(* Logix 5000 project; controller cal1615 1756-L62 rev 16.20; software revision 16.05; part 58 of 78 *)
(* tags used below, declared in another part *)
   FAULT : BOOL;   // Fault AFI
   HMI : BOOL;   // AFI HMI
   p01r09_pb_global_reset : BOOL;   // System Modes PB: Global Fault Reset
   p02_real_from_hmi : hmi_real;   // MOP HMI Iface Real from HMI
   p25_ai_amps : DINT;   // Tension Stand 2 Analog Input TS 2 Motor Current
   p25_ai_hz : DINT;   // Tension Stand 2 Analog Input TS 2 Motor Hertz
   p25_ai_rpm : REAL;
   p25_ai_speed : REAL;   // Tension Stand 2 Inputs Sufrace Speed [fpm]
   p25_ai_ts2_lc : REAL;   // System Metering Roll VFD Minimum Start Tension
   p25_ao_selected_speed : REAL;   // Tension Stand 2 VFD Selected Speed
   p25_ao_torque : REAL;
   p25_ao_vfd : REAL;
   p25_control_word : INT;
   p25_di_brake : BOOL;   // Tension Stand 2 Digital Input TS2 & Slitter Brake Temperature OK
   p25_di_therm : BOOL;   // Tension Stand 2 Digital Input Motor Temperature OK
   p25_di_ts2 : acs800_di_normal;   // Tension Stand 2 Digital Inputs VFD Inputs
   p25_dint_to_hmi : DINT[16];   // Tension Stand 2 Dint to HMI
   p25_real_to_hmi : REAL[112];   // Tension Stand 2 Real to HMI
   p25_status_word : INT;
   p25_ts2_gear_ratio : REAL;
   p25_ts2_roll_diameter_ft : REAL;
   p25_vfd_input_max : REAL;
   p25_vfd_input_min : REAL;
   p25_vfd_output_max : REAL;
   p25_vfd_output_min : REAL;
   p25r01 : routine;
   p25r03_vfd_out_scaling : SYS_SCP;
   p25r04 : routine;
   p25r04_speed_to_vfd_ts2_scp : SYS_SPEED_TO_VFD;   // Tension Stand 2 Outputs Speed to Tension Stand 2 VFD
   p25r04_timer_fault : TIMER[4];   // Tension Stand 2 Outputs Fault Dwell Timer
   p25r04_timer_warning : TIMER[4];   // Tension Stand 2 Outputs Warning Dwell Timer
   p25r05 : routine;
   p25r05_timer_fault : TIMER[4];   // Tension Stand 2 Dint to HMI Fault Dwell Timer
   p25r05_timer_warning : TIMER[4];   // Tension Stand 2 Dint to HMI Warning Dwell Time
   p25r06 : routine;
   p25r06_ave_lc : REAL;
   p25r06_lc_ave_ctrl : CONTROL;
   p25r06_lc_buffer : REAL[20];
   p25r06_lc_ctrl : CONTROL;
   p25r06_sample_timer : TIMER;
   p25r06_timer_fault : TIMER[4];   // Tension Stand 2 Real to HMI Fault Dwell Timer
   p25r06_timer_warning : TIMER[4];   // Tension Stand 2 Real to HMI Warning Dwell Timer
   p25r06_unload : REAL;
   p25r09_mode_jog : BOOL;   // Tension Stand 2 Modes Jog Mode
   p25r09_mode_run : BOOL;   // Tension Stand 2 Modes Run Mode
   p25r09_mode_thread : BOOL;   // Tension Stand 2 Modes Thread Mode
(* P25_Tension_Stand_2, continued *)

ROUTINE R04_Output   (* ladder *)
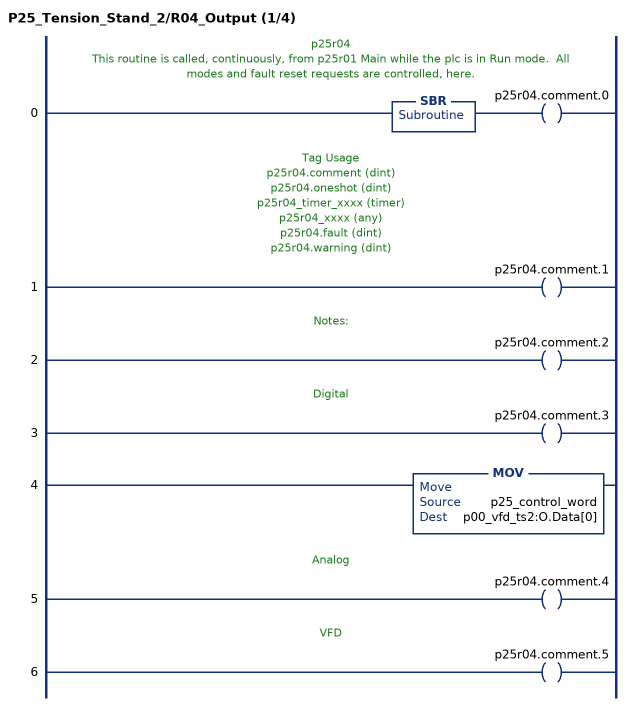
   // p25r04
   // This routine is called, continuously, from p25r01 Main while the plc is in Run mode.  All modes and fault reset requests are controlled, here.
   0: SBR()OTE(p25r04.comment.0);
   // Tag Usage
   // p25r04.comment (dint)
   // p25r04.oneshot (dint)
   // p25r04_timer_xxxx (timer)
   // p25r04_xxxx (any)
   // p25r04.fault (dint)
   // p25r04.warning (dint)
   1: OTE(p25r04.comment.1);
   // Notes:
   2: OTE(p25r04.comment.2);
   // Digital
   3: OTE(p25r04.comment.3);
   4: MOV(p25_control_word,p00_vfd_ts2:O.Data[0]);
   // Analog
   5: OTE(p25r04.comment.4);
   // VFD
   6: OTE(p25r04.comment.5);
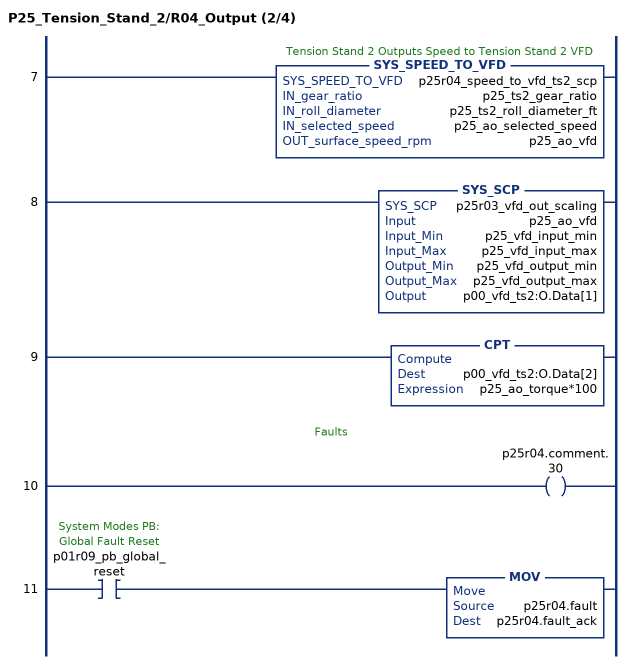
   7: SYS_SPEED_TO_VFD(p25r04_speed_to_vfd_ts2_scp,p25_ts2_gear_ratio,p25_ts2_roll_diameter_ft,p25_ao_selected_speed,p25_ao_vfd);
   8: SYS_SCP(p25r03_vfd_out_scaling,p25_ao_vfd,p25_vfd_input_min,p25_vfd_input_max,p25_vfd_output_min,p25_vfd_output_max,p00_vfd_ts2:O.Data[1]);
   9: CPT(p00_vfd_ts2:O.Data[2],p25_ao_torque*100);
   // Faults
   10: OTE(p25r04.comment.30);
   11: XIC(p01r09_pb_global_reset)MOV(p25r04.fault,p25r04.fault_ack);
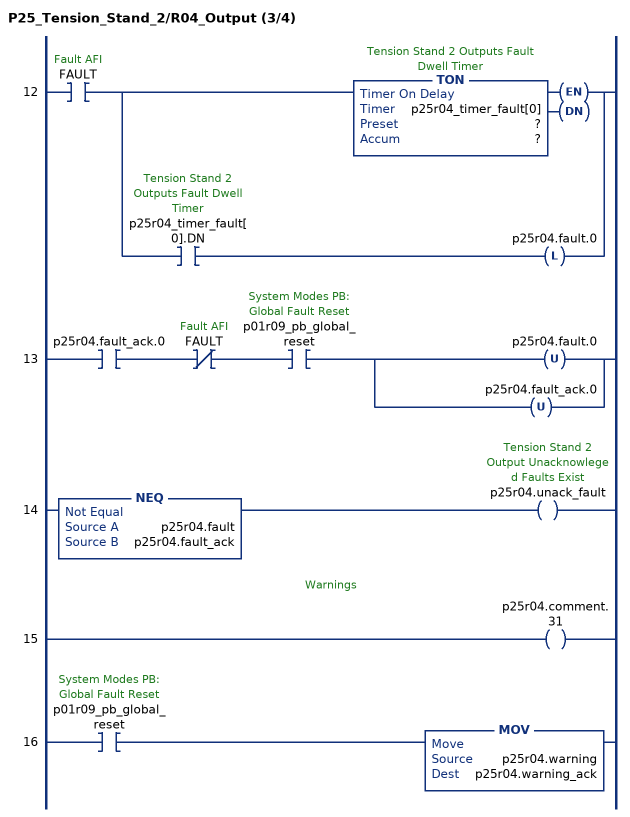
   12: XIC(FAULT)[TON(p25r04_timer_fault[0],?,?) ,XIC(p25r04_timer_fault[0].DN) OTL(p25r04.fault.0) ];
   13: XIC(p25r04.fault_ack.0)XIO(FAULT)XIC(p01r09_pb_global_reset)[OTU(p25r04.fault.0) ,OTU(p25r04.fault_ack.0) ];
   14: NEQ(p25r04.fault,p25r04.fault_ack)OTE(p25r04.unack_fault);
   // Warnings
   15: OTE(p25r04.comment.31);
   16: XIC(p01r09_pb_global_reset)MOV(p25r04.warning,p25r04.warning_ack);
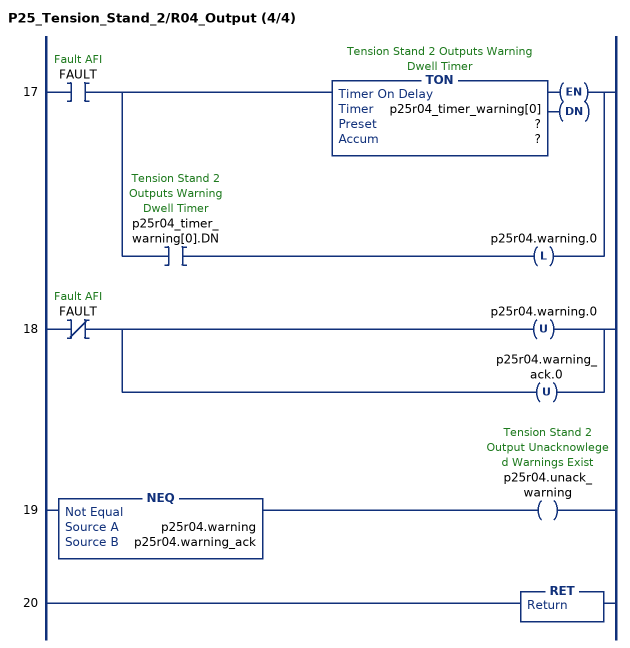
   17: XIC(FAULT)[TON(p25r04_timer_warning[0],?,?) ,XIC(p25r04_timer_warning[0].DN) OTL(p25r04.warning.0) ];
   18: XIO(FAULT)[OTU(p25r04.warning.0) ,OTU(p25r04.warning_ack.0) ];
   19: NEQ(p25r04.warning,p25r04.warning_ack)OTE(p25r04.unack_warning);
   20: RET();
END_ROUTINE

ROUTINE R05_Dint_to_HMI   (* ladder *)
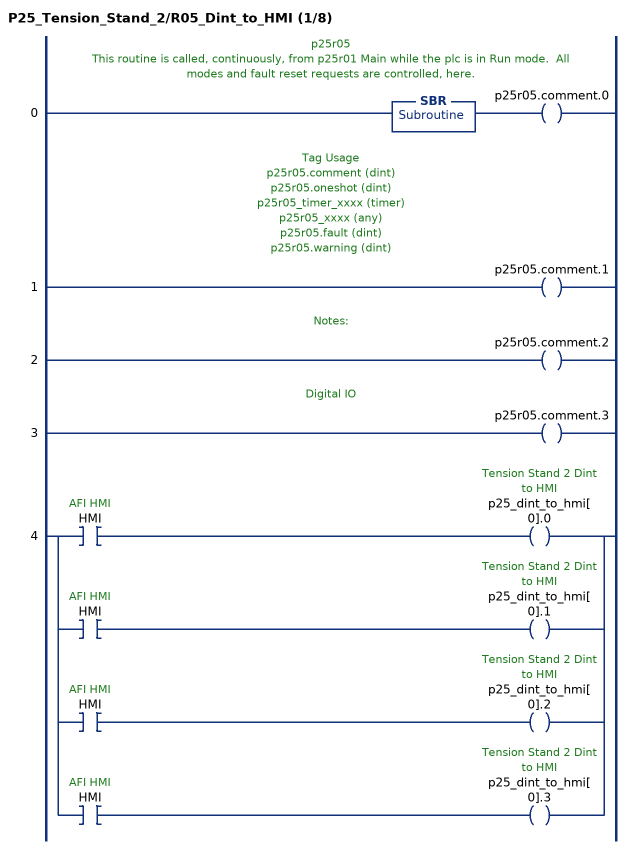
   // p25r05
   // This routine is called, continuously, from p25r01 Main while the plc is in Run mode.  All modes and fault reset requests are controlled, here.
   0: SBR()OTE(p25r05.comment.0);
   // Tag Usage
   // p25r05.comment (dint)
   // p25r05.oneshot (dint)
   // p25r05_timer_xxxx (timer)
   // p25r05_xxxx (any)
   // p25r05.fault (dint)
   // p25r05.warning (dint)
   1: OTE(p25r05.comment.1);
   // Notes:
   2: OTE(p25r05.comment.2);
   // Digital IO
   3: OTE(p25r05.comment.3);
   4: [XIC(HMI) OTE(p25_dint_to_hmi[0].0) ,XIC(HMI) OTE(p25_dint_to_hmi[0].1) ,XIC(HMI) OTE(p25_dint_to_hmi[0].2) ,XIC(HMI) OTE(p25_dint_to_hmi[0].3) ];
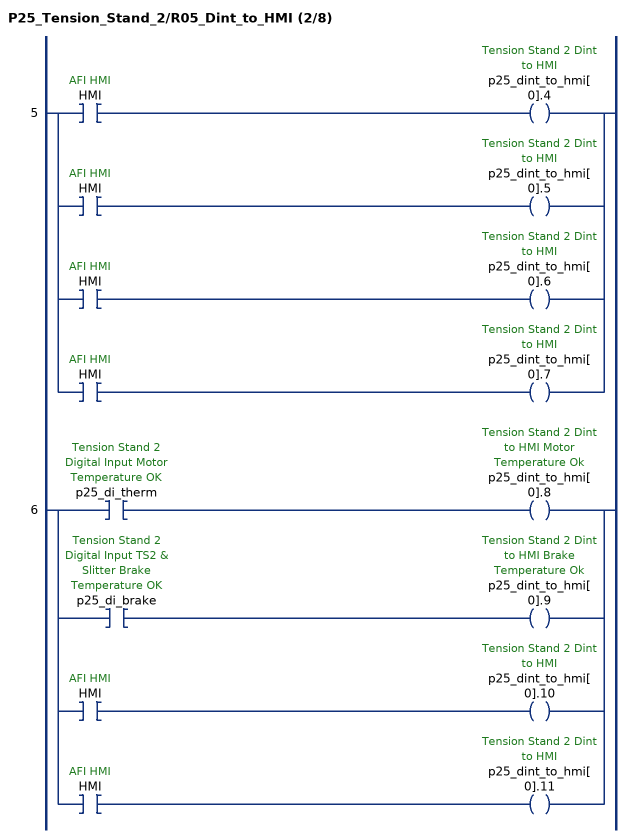
   5: [XIC(HMI) OTE(p25_dint_to_hmi[0].4) ,XIC(HMI) OTE(p25_dint_to_hmi[0].5) ,XIC(HMI) OTE(p25_dint_to_hmi[0].6) ,XIC(HMI) OTE(p25_dint_to_hmi[0].7) ];
   6: [XIC(p25_di_therm) OTE(p25_dint_to_hmi[0].8) ,XIC(p25_di_brake) OTE(p25_dint_to_hmi[0].9) ,XIC(HMI) OTE(p25_dint_to_hmi[0].10) ,XIC(HMI) OTE(p25_dint_to_hmi[0].11) ];
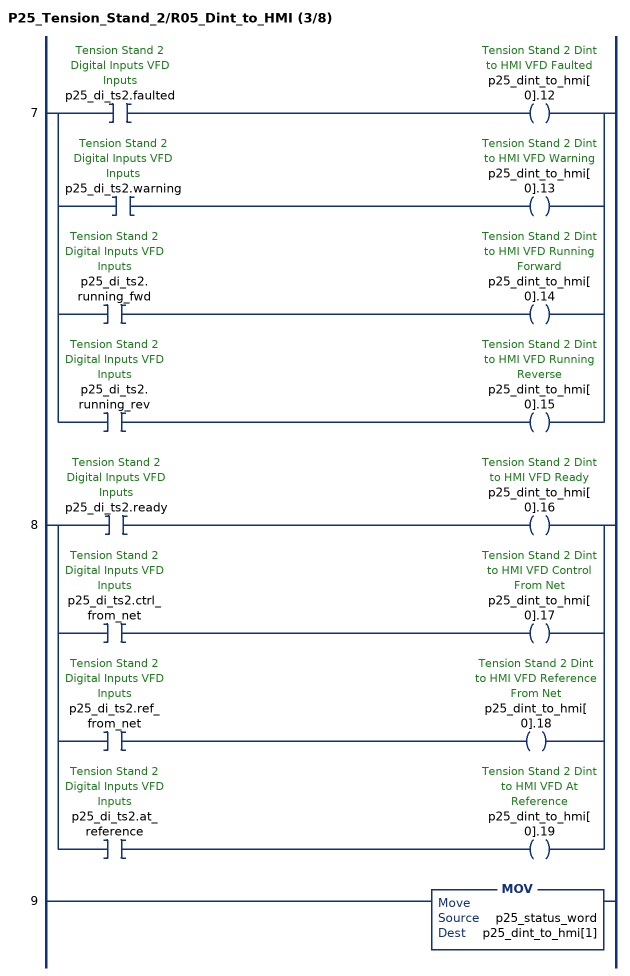
   7: [XIC(p25_di_ts2.faulted) OTE(p25_dint_to_hmi[0].12) ,XIC(p25_di_ts2.warning) OTE(p25_dint_to_hmi[0].13) ,XIC(p25_di_ts2.running_fwd) OTE(p25_dint_to_hmi[0].14) ,XIC(p25_di_ts2.running_rev) OTE(p25_dint_to_hmi[0].15) ];
   8: [XIC(p25_di_ts2.ready) OTE(p25_dint_to_hmi[0].16) ,XIC(p25_di_ts2.ctrl_from_net) OTE(p25_dint_to_hmi[0].17) ,XIC(p25_di_ts2.ref_from_net) OTE(p25_dint_to_hmi[0].18) ,XIC(p25_di_ts2.at_reference) OTE(p25_dint_to_hmi[0].19) ];
   9: MOV(p25_status_word,p25_dint_to_hmi[1]);
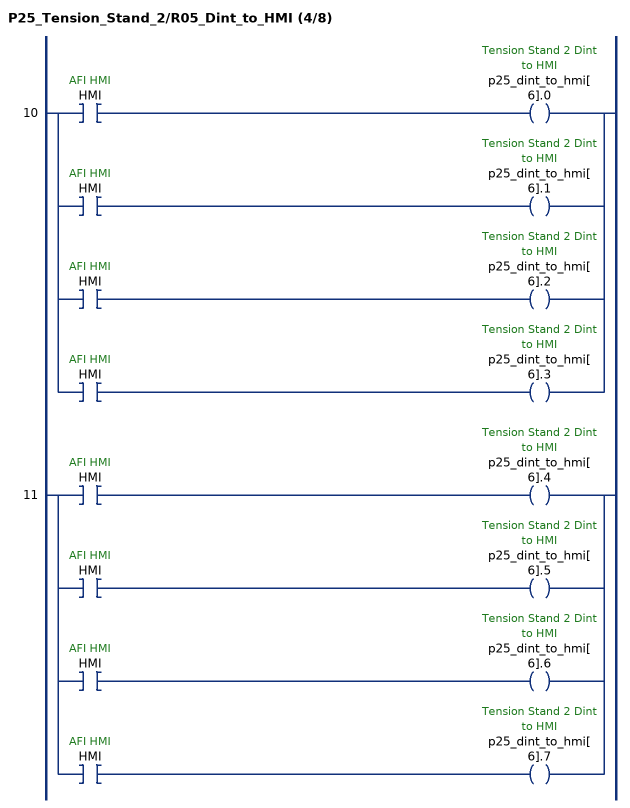
   10: [XIC(HMI) OTE(p25_dint_to_hmi[6].0) ,XIC(HMI) OTE(p25_dint_to_hmi[6].1) ,XIC(HMI) OTE(p25_dint_to_hmi[6].2) ,XIC(HMI) OTE(p25_dint_to_hmi[6].3) ];
   11: [XIC(HMI) OTE(p25_dint_to_hmi[6].4) ,XIC(HMI) OTE(p25_dint_to_hmi[6].5) ,XIC(HMI) OTE(p25_dint_to_hmi[6].6) ,XIC(HMI) OTE(p25_dint_to_hmi[6].7) ];
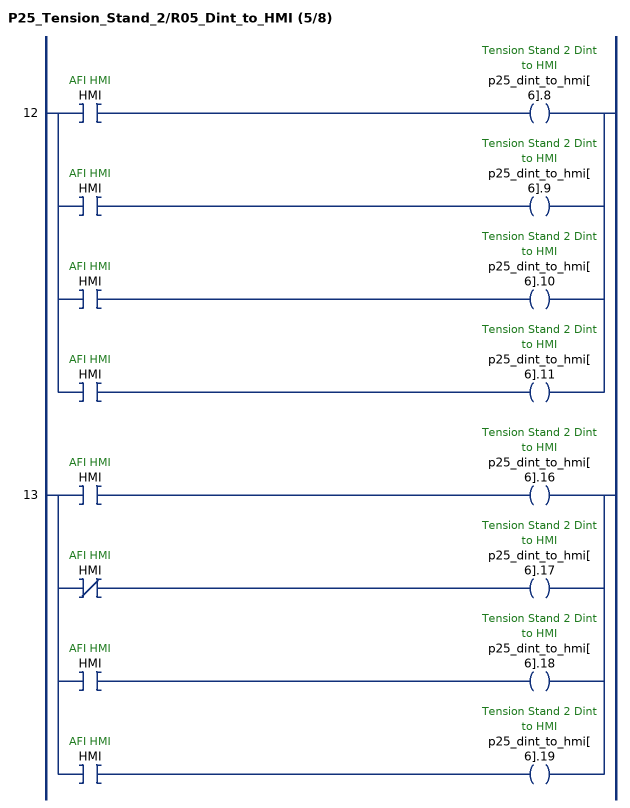
   12: [XIC(HMI) OTE(p25_dint_to_hmi[6].8) ,XIC(HMI) OTE(p25_dint_to_hmi[6].9) ,XIC(HMI) OTE(p25_dint_to_hmi[6].10) ,XIC(HMI) OTE(p25_dint_to_hmi[6].11) ];
   13: [XIC(HMI) OTE(p25_dint_to_hmi[6].16) ,XIO(HMI) OTE(p25_dint_to_hmi[6].17) ,XIC(HMI) OTE(p25_dint_to_hmi[6].18) ,XIC(HMI) OTE(p25_dint_to_hmi[6].19) ];
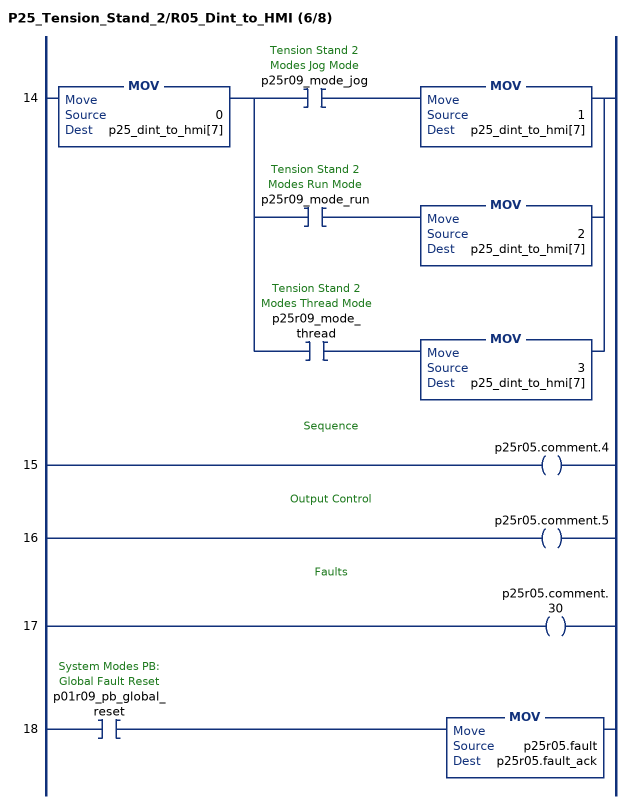
   14: MOV(0,p25_dint_to_hmi[7])[XIC(p25r09_mode_jog) MOV(1,p25_dint_to_hmi[7]) ,XIC(p25r09_mode_run) MOV(2,p25_dint_to_hmi[7]) ,XIC(p25r09_mode_thread) MOV(3,p25_dint_to_hmi[7]) ];
   // Sequence
   15: OTE(p25r05.comment.4);
   // Output Control
   16: OTE(p25r05.comment.5);
   // Faults
   17: OTE(p25r05.comment.30);
   18: XIC(p01r09_pb_global_reset)MOV(p25r05.fault,p25r05.fault_ack);
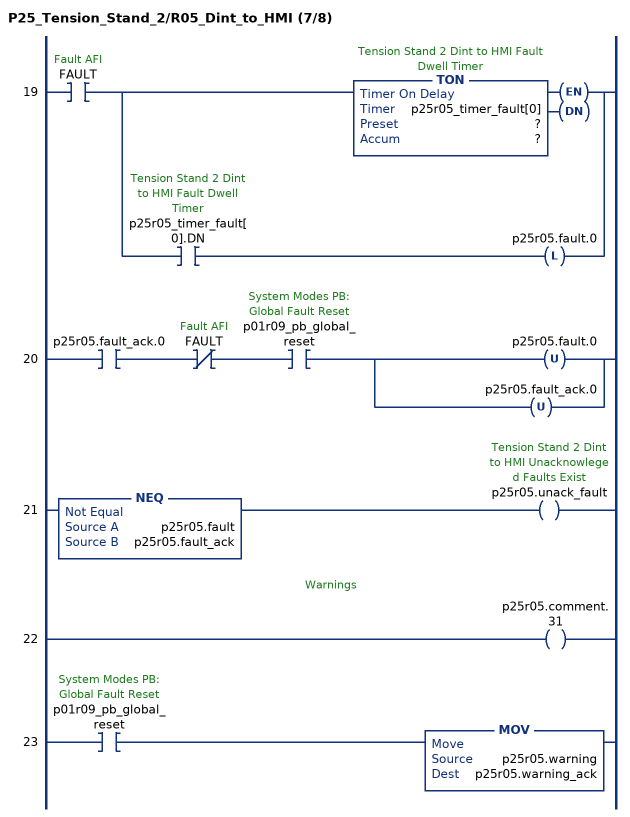
   19: XIC(FAULT)[TON(p25r05_timer_fault[0],?,?) ,XIC(p25r05_timer_fault[0].DN) OTL(p25r05.fault.0) ];
   20: XIC(p25r05.fault_ack.0)XIO(FAULT)XIC(p01r09_pb_global_reset)[OTU(p25r05.fault.0) ,OTU(p25r05.fault_ack.0) ];
   21: NEQ(p25r05.fault,p25r05.fault_ack)OTE(p25r05.unack_fault);
   // Warnings
   22: OTE(p25r05.comment.31);
   23: XIC(p01r09_pb_global_reset)MOV(p25r05.warning,p25r05.warning_ack);
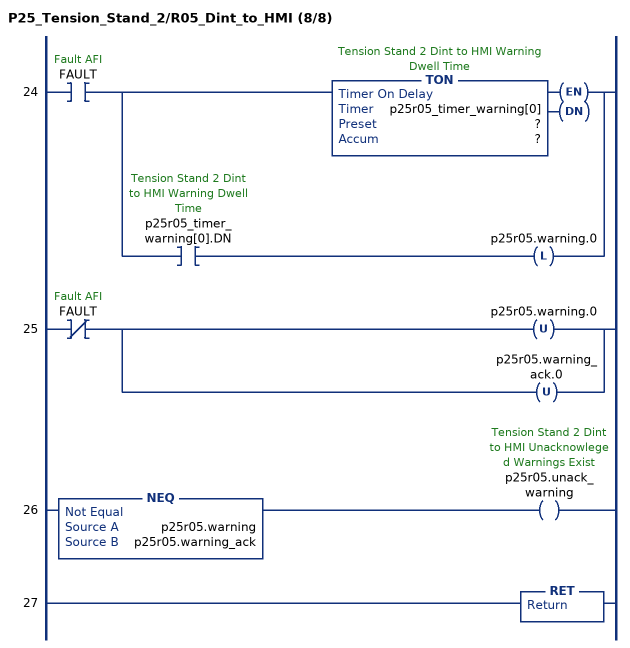
   24: XIC(FAULT)[TON(p25r05_timer_warning[0],?,?) ,XIC(p25r05_timer_warning[0].DN) OTL(p25r05.warning.0) ];
   25: XIO(FAULT)[OTU(p25r05.warning.0) ,OTU(p25r05.warning_ack.0) ];
   26: NEQ(p25r05.warning,p25r05.warning_ack)OTE(p25r05.unack_warning);
   27: RET();
END_ROUTINE

ROUTINE R06_Real_to_HMI   (* ladder *)
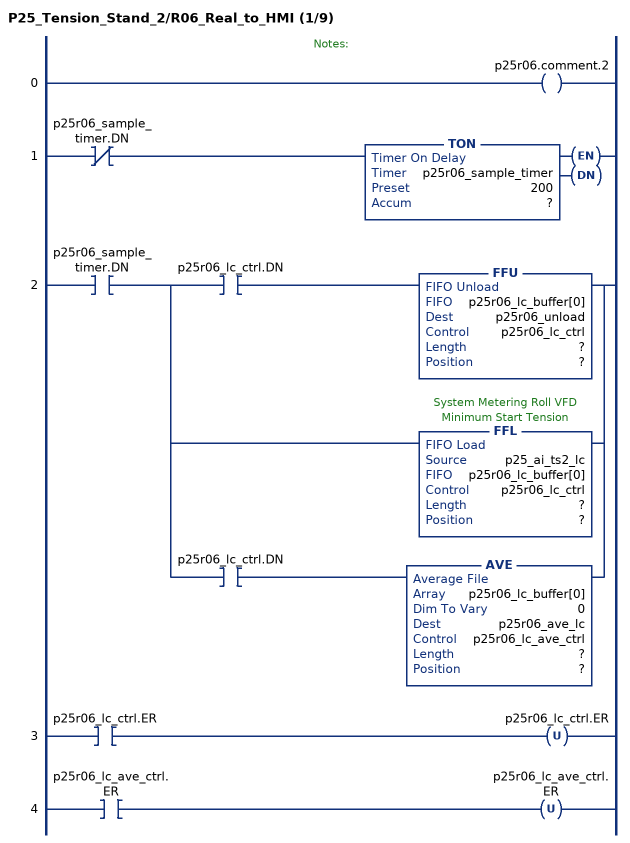
   // Notes:
   0: OTE(p25r06.comment.2);
   1: XIO(p25r06_sample_timer.DN)TON(p25r06_sample_timer,?,?);
   2: XIC(p25r06_sample_timer.DN)[XIC(p25r06_lc_ctrl.DN) FFU(p25r06_lc_buffer[0],p25r06_unload,p25r06_lc_ctrl,?,?) ,FFL(p25_ai_ts2_lc,p25r06_lc_buffer[0],p25r06_lc_ctrl,?,?) ,XIC(p25r06_lc_ctrl.DN) AVE(p25r06_lc_buffer[0],0,p25r06_ave_lc,p25r06_lc_ave_ctrl,?,?) ];
   3: XIC(p25r06_lc_ctrl.ER)OTU(p25r06_lc_ctrl.ER);
   4: XIC(p25r06_lc_ave_ctrl.ER)OTU(p25r06_lc_ave_ctrl.ER);
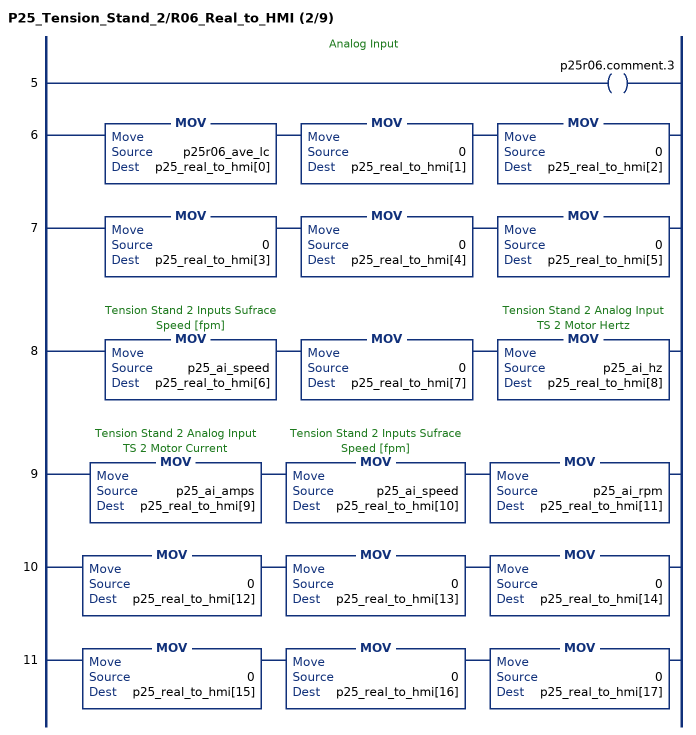
   // Analog Input
   5: OTE(p25r06.comment.3);
   6: MOV(p25r06_ave_lc,p25_real_to_hmi[0])MOV(0,p25_real_to_hmi[1])MOV(0,p25_real_to_hmi[2]);
   7: MOV(0,p25_real_to_hmi[3])MOV(0,p25_real_to_hmi[4])MOV(0,p25_real_to_hmi[5]);
   8: MOV(p25_ai_speed,p25_real_to_hmi[6])MOV(0,p25_real_to_hmi[7])MOV(p25_ai_hz,p25_real_to_hmi[8]);
   9: MOV(p25_ai_amps,p25_real_to_hmi[9])MOV(p25_ai_speed,p25_real_to_hmi[10])MOV(p25_ai_rpm,p25_real_to_hmi[11]);
   10: MOV(0,p25_real_to_hmi[12])MOV(0,p25_real_to_hmi[13])MOV(0,p25_real_to_hmi[14]);
   11: MOV(0,p25_real_to_hmi[15])MOV(0,p25_real_to_hmi[16])MOV(0,p25_real_to_hmi[17]);
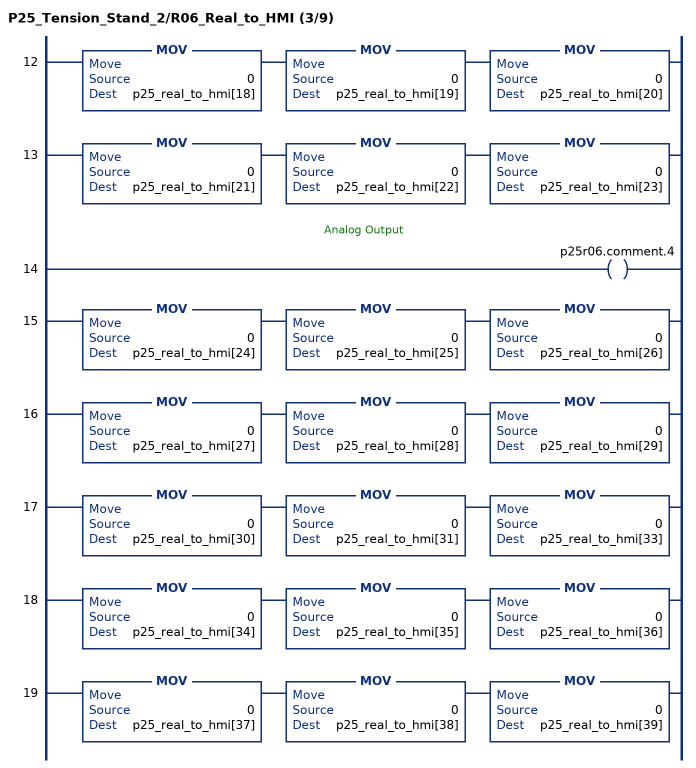
   12: MOV(0,p25_real_to_hmi[18])MOV(0,p25_real_to_hmi[19])MOV(0,p25_real_to_hmi[20]);
   13: MOV(0,p25_real_to_hmi[21])MOV(0,p25_real_to_hmi[22])MOV(0,p25_real_to_hmi[23]);
   // Analog Output
   14: OTE(p25r06.comment.4);
   15: MOV(0,p25_real_to_hmi[24])MOV(0,p25_real_to_hmi[25])MOV(0,p25_real_to_hmi[26]);
   16: MOV(0,p25_real_to_hmi[27])MOV(0,p25_real_to_hmi[28])MOV(0,p25_real_to_hmi[29]);
   17: MOV(0,p25_real_to_hmi[30])MOV(0,p25_real_to_hmi[31])MOV(0,p25_real_to_hmi[33]);
   18: MOV(0,p25_real_to_hmi[34])MOV(0,p25_real_to_hmi[35])MOV(0,p25_real_to_hmi[36]);
   19: MOV(0,p25_real_to_hmi[37])MOV(0,p25_real_to_hmi[38])MOV(0,p25_real_to_hmi[39]);
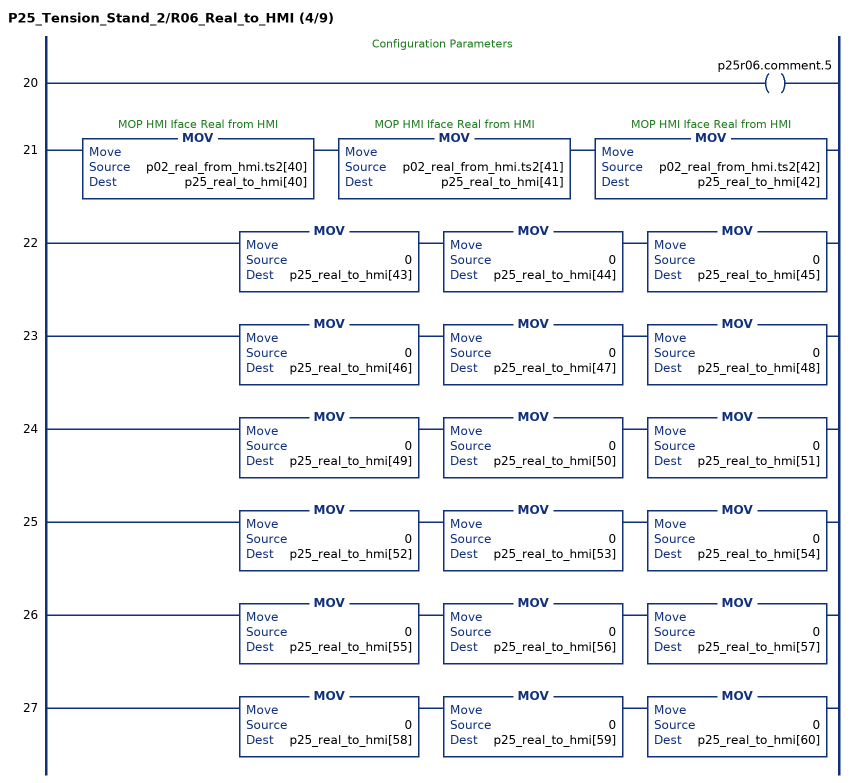
   // Configuration Parameters
   20: OTE(p25r06.comment.5);
   21: MOV(p02_real_from_hmi.ts2[40],p25_real_to_hmi[40])MOV(p02_real_from_hmi.ts2[41],p25_real_to_hmi[41])MOV(p02_real_from_hmi.ts2[42],p25_real_to_hmi[42]);
   22: MOV(0,p25_real_to_hmi[43])MOV(0,p25_real_to_hmi[44])MOV(0,p25_real_to_hmi[45]);
   23: MOV(0,p25_real_to_hmi[46])MOV(0,p25_real_to_hmi[47])MOV(0,p25_real_to_hmi[48]);
   24: MOV(0,p25_real_to_hmi[49])MOV(0,p25_real_to_hmi[50])MOV(0,p25_real_to_hmi[51]);
   25: MOV(0,p25_real_to_hmi[52])MOV(0,p25_real_to_hmi[53])MOV(0,p25_real_to_hmi[54]);
   26: MOV(0,p25_real_to_hmi[55])MOV(0,p25_real_to_hmi[56])MOV(0,p25_real_to_hmi[57]);
   27: MOV(0,p25_real_to_hmi[58])MOV(0,p25_real_to_hmi[59])MOV(0,p25_real_to_hmi[60]);
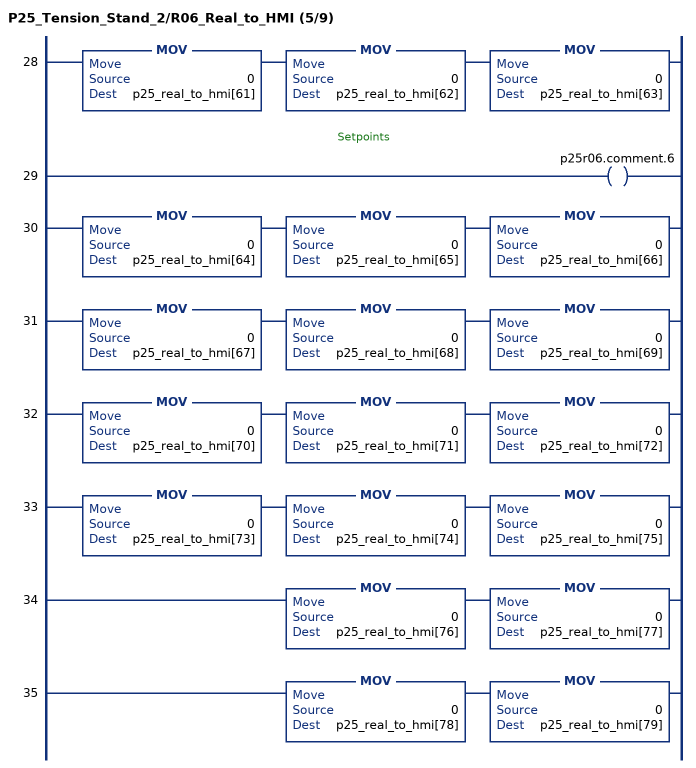
   28: MOV(0,p25_real_to_hmi[61])MOV(0,p25_real_to_hmi[62])MOV(0,p25_real_to_hmi[63]);
   // Setpoints
   29: OTE(p25r06.comment.6);
   30: MOV(0,p25_real_to_hmi[64])MOV(0,p25_real_to_hmi[65])MOV(0,p25_real_to_hmi[66]);
   31: MOV(0,p25_real_to_hmi[67])MOV(0,p25_real_to_hmi[68])MOV(0,p25_real_to_hmi[69]);
   32: MOV(0,p25_real_to_hmi[70])MOV(0,p25_real_to_hmi[71])MOV(0,p25_real_to_hmi[72]);
   33: MOV(0,p25_real_to_hmi[73])MOV(0,p25_real_to_hmi[74])MOV(0,p25_real_to_hmi[75]);
   34: MOV(0,p25_real_to_hmi[76])MOV(0,p25_real_to_hmi[77]);
   35: MOV(0,p25_real_to_hmi[78])MOV(0,p25_real_to_hmi[79]);
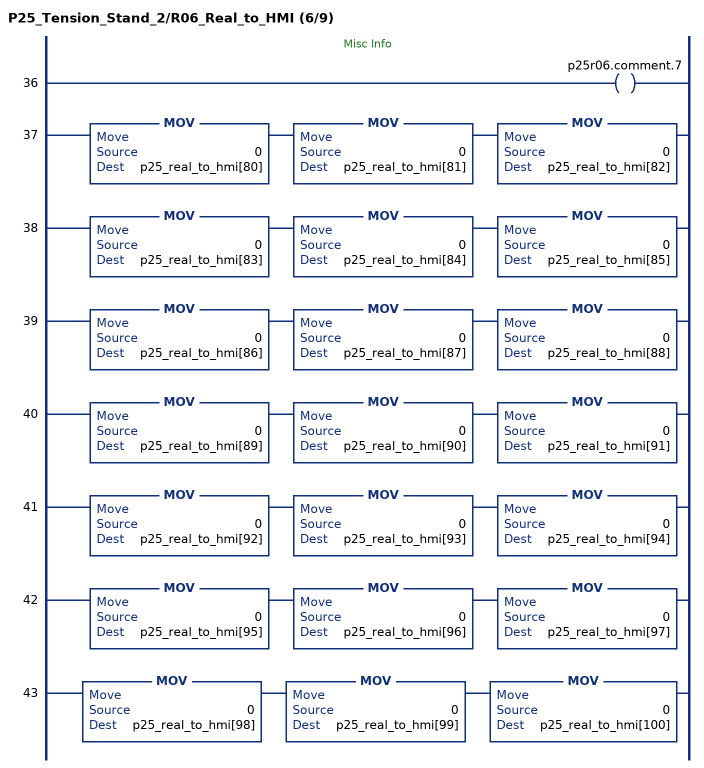
   // Misc Info
   36: OTE(p25r06.comment.7);
   37: MOV(0,p25_real_to_hmi[80])MOV(0,p25_real_to_hmi[81])MOV(0,p25_real_to_hmi[82]);
   38: MOV(0,p25_real_to_hmi[83])MOV(0,p25_real_to_hmi[84])MOV(0,p25_real_to_hmi[85]);
   39: MOV(0,p25_real_to_hmi[86])MOV(0,p25_real_to_hmi[87])MOV(0,p25_real_to_hmi[88]);
   40: MOV(0,p25_real_to_hmi[89])MOV(0,p25_real_to_hmi[90])MOV(0,p25_real_to_hmi[91]);
   41: MOV(0,p25_real_to_hmi[92])MOV(0,p25_real_to_hmi[93])MOV(0,p25_real_to_hmi[94]);
   42: MOV(0,p25_real_to_hmi[95])MOV(0,p25_real_to_hmi[96])MOV(0,p25_real_to_hmi[97]);
   43: MOV(0,p25_real_to_hmi[98])MOV(0,p25_real_to_hmi[99])MOV(0,p25_real_to_hmi[100]);
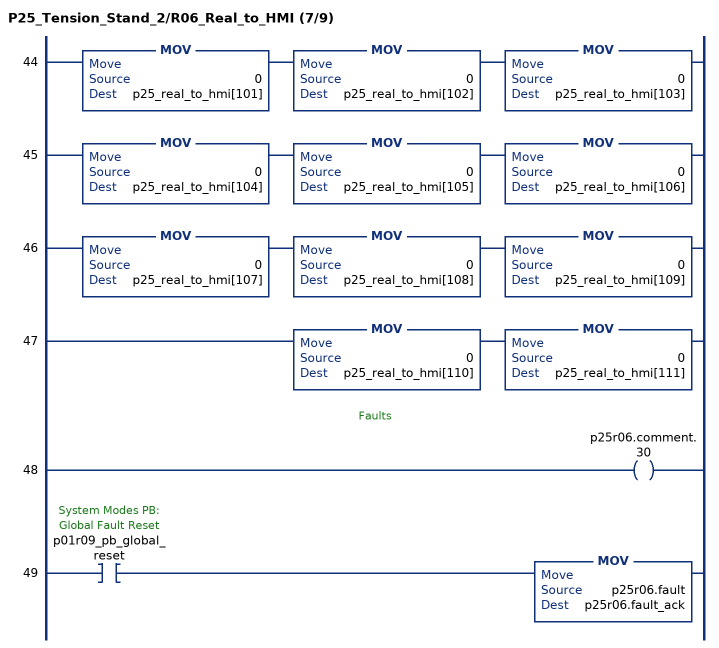
   44: MOV(0,p25_real_to_hmi[101])MOV(0,p25_real_to_hmi[102])MOV(0,p25_real_to_hmi[103]);
   45: MOV(0,p25_real_to_hmi[104])MOV(0,p25_real_to_hmi[105])MOV(0,p25_real_to_hmi[106]);
   46: MOV(0,p25_real_to_hmi[107])MOV(0,p25_real_to_hmi[108])MOV(0,p25_real_to_hmi[109]);
   47: MOV(0,p25_real_to_hmi[110])MOV(0,p25_real_to_hmi[111]);
   // Faults
   48: OTE(p25r06.comment.30);
   49: XIC(p01r09_pb_global_reset)MOV(p25r06.fault,p25r06.fault_ack);
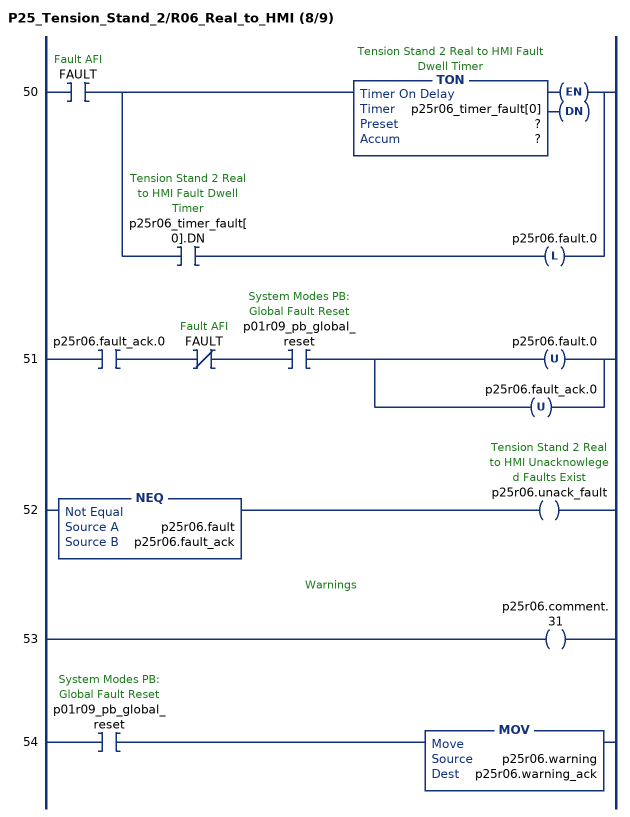
   50: XIC(FAULT)[TON(p25r06_timer_fault[0],?,?) ,XIC(p25r06_timer_fault[0].DN) OTL(p25r06.fault.0) ];
   51: XIC(p25r06.fault_ack.0)XIO(FAULT)XIC(p01r09_pb_global_reset)[OTU(p25r06.fault.0) ,OTU(p25r06.fault_ack.0) ];
   52: NEQ(p25r06.fault,p25r06.fault_ack)OTE(p25r06.unack_fault);
   // Warnings
   53: OTE(p25r06.comment.31);
   54: XIC(p01r09_pb_global_reset)MOV(p25r06.warning,p25r06.warning_ack);
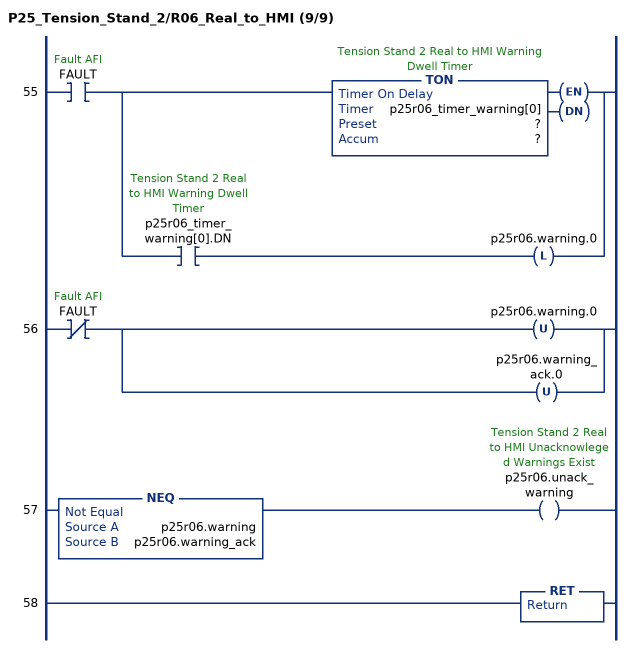
   55: XIC(FAULT)[TON(p25r06_timer_warning[0],?,?) ,XIC(p25r06_timer_warning[0].DN) OTL(p25r06.warning.0) ];
   56: XIO(FAULT)[OTU(p25r06.warning.0) ,OTU(p25r06.warning_ack.0) ];
   57: NEQ(p25r06.warning,p25r06.warning_ack)OTE(p25r06.unack_warning);
   58: RET();
END_ROUTINE
